FUNCTION_BLOCK Day
VAR_INPUT
	
END_VAR
VAR_OUTPUT
END_VAR
VAR
END_VAR

END_FUNCTION_BLOCK

(* stored: Version 1.1.0.1, ProductVersion 3.1.4024.12
   POU Day: Id {2917063c-683d-4163-b0a5-9371e8d60321}, SpecialFunc None *)
